# EPICS substitutions: evrSupport/Db/bsa/bsaFARCEdef.substitutions
#==============================================================================
#
# Abs:  Beam Synchronous Acquisition records for a single Toroid.
#
# Name: bsaFARCEdef.substitutions
#
# Note: Must follow the LCLS naming conventions.
#
#==============================================================================
# BSA Integration Note:
# Each device attribute (such as width ) provides input to bsaEdefAvg.db.
# The bsaEdefAvg.db provides the RMS and Avg -$(DEV):$(SECN)<edef id>, and history -
#   $(DEV):$(SECN)HST<edef id> for each device attribute for each of 20 edefs.
#
file bsaEdefAvg.db
{
#	      Device           Name                                      IOC    IOC   mod5  Init
#                                                                    loc'n  unit  bit   Event Code
  pattern {DEV    ,SECN, INP           , DESC  , MD,MDID, EGU ,HOPR  ,LOPR  ,PREC, ADEL, MDEL  , LOCA  , UNIT ,BIT, EC}
	  { $(DEVICE) ,CHRG, $(DEVICE):CHRG,  1    , 1,  1  , ""  ,"3E10","1E10",  3 ,"1E8","1E7"  , $(LOC), $(UN), A, 101}
	  { $(DEVICE) ,CHRG, $(DEVICE):CHRG,  2    , 2,  2  , ""  ,"3E10","1E10",  3 ,"1E8","1E7"  , $(LOC), $(UN), B, 102}
	  { $(DEVICE) ,CHRG, $(DEVICE):CHRG,  3    , 3,  3  , ""  ,"3E10","1E10",  3 ,"1E8","1E7"  , $(LOC), $(UN), C, 103}
	  { $(DEVICE) ,CHRG, $(DEVICE):CHRG,  4    , 4,  4  , ""  ,"3E10","1E10",  3 ,"1E8","1E7"  , $(LOC), $(UN), D, 104}
	  { $(DEVICE) ,CHRG, $(DEVICE):CHRG,  5    , 5,  5  , ""  ,"3E10","1E10",  3 ,"1E8","1E7"  , $(LOC), $(UN), E, 105}
	  { $(DEVICE) ,CHRG, $(DEVICE):CHRG,  6    , 6,  6  , ""  ,"3E10","1E10",  3 ,"1E8","1E7"  , $(LOC), $(UN), F, 106}
	  { $(DEVICE) ,CHRG, $(DEVICE):CHRG,  7    , 7,  7  , ""  ,"3E10","1E10",  3 ,"1E8","1E7"  , $(LOC), $(UN), G, 107}
	  { $(DEVICE) ,CHRG, $(DEVICE):CHRG,  8    , 8,  8  , ""  ,"3E10","1E10",  3 ,"1E8","1E7"  , $(LOC), $(UN), H, 108}
	  { $(DEVICE) ,CHRG, $(DEVICE):CHRG,  9    , 9,  9  , ""  ,"3E10","1E10",  3 ,"1E8","1E7"  , $(LOC), $(UN), I, 109}
	  { $(DEVICE) ,CHRG, $(DEVICE):CHRG,  10   ,10,  10 , ""  ,"3E10","1E10",  3 ,"1E8","1E7"  , $(LOC), $(UN), J, 110}
	  { $(DEVICE) ,CHRG, $(DEVICE):CHRG,  11   ,11,  11 , ""  ,"3E10","1E10",  3 ,"1E8","1E7"  , $(LOC), $(UN), K, 111}
	  { $(DEVICE) ,CHRG, $(DEVICE):CHRG,  12   ,12,  12 , ""  ,"3E10","1E10",  3 ,"1E8","1E7"  , $(LOC), $(UN), L, 112}
	  { $(DEVICE) ,CHRG, $(DEVICE):CHRG,  13   ,13,  13 , ""  ,"3E10","1E10",  3 ,"1E8","1E7"  , $(LOC), $(UN), M, 113}
	  { $(DEVICE) ,CHRG, $(DEVICE):CHRG,  14   ,14,  14 , ""  ,"3E10","1E10",  3 ,"1E8","1E7"  , $(LOC), $(UN), N, 114}
	  { $(DEVICE) ,CHRG, $(DEVICE):CHRG,  15   ,15,  15 , ""  ,"3E10","1E10",  3 ,"1E8","1E7"  , $(LOC), $(UN), O, 115}
	  { $(DEVICE) ,CHRG, $(DEVICE):CHRG,  1HZ  ,16,  1H , ""  ,"3E10","1E10",  3 ,"1E8","1E7"  , $(LOC), $(UN), P, 116}
	  { $(DEVICE) ,CHRG, $(DEVICE):CHRG,  10HZ ,17,  TH , ""  ,"3E10","1E10",  3 ,"1E8","1E7"  , $(LOC), $(UN), Q, 117}
	  { $(DEVICE) ,CHRG, $(DEVICE):CHRG,  FULL ,18,  BR , ""  ,"3E10","1E10",  3 ,"1E8","1E7"  , $(LOC), $(UN), R, 118}
	  { $(DEVICE) ,CHRG, $(DEVICE):CHRG,  FBCK1,19,  F1 , ""  ,"3E10","1E10",  3 ,"1E8","1E7"  , $(LOC), $(UN), S, 119}
	  { $(DEVICE) ,CHRG, $(DEVICE):CHRG,  FBCK2,20,  F2 , ""  ,"3E10","1E10",  3 ,"1E8","1E7"  , $(LOC), $(UN), T, 120}
}

file bsaEdefFanouts.db
{
#	      Device           Name
  pattern {DEV    ,SECN , FLNK }
	  { $(DEVICE) ,CHRG ,  ""  }
}
